PROGRAM PRG_OpcuaMonitor

VAR_OUTPUT
	Error : BOOL;	
END_VAR
VAR
	fbFCUHb	: FB_HeartbeatMonitor;
	fbSpindleHb	: FB_HeartbeatMonitor;
END_VAR

Error := FALSE;

fbFCUHb(CLK:= GVL_opcua.stFcuControl.status.input.Heartbeat, T:= T#2.5S, Q=> );
IF NOT fbFCUHb.Q THEN
	// There's no way to simply disable the fcu.  
	GVL_opcua.stFcuControl.input.SetControlMode := E_FCU_ControlMode.SoftTouch;
	GVL_opcua.stFcuControl.input.SetForce := 0;	
	Error := TRUE;
ELSE
	Error := FALSE;
END_IF



fbSpindleHb(CLK:= GVL_opcua.stSpindleControl.status.input.Heartbeat, T:= T#2.5S, Q=> );
IF NOT fbSpindleHb.Q THEN
	MEMSET(ADR(GVL_opcua.stSpindleControl.input), 0, SIZEOF(GVL_opcua.stSpindleControl.input));
	Error := TRUE;
ELSE
	Error := FALSE;
END_IF

END_PROGRAM

(* stored: Version 1.1.0.1, ProductVersion 3.1.4024.9
   POU PRG_OpcuaMonitor: Id {d8833ab7-3197-4713-a10b-d7af028115a9}, SpecialFunc None *)
